FUNCTION_BLOCK FB_Component_SingleValve IMPLEMENTS I_Component
VAR_INPUT
	sName			: STRING[50];
	tTimeout		: TIME := T#0S;
END_VAR

VAR_IN_OUT
	bOutput			: BOOL;
END_VAR

VAR_OUTPUT
	bEnabled     	: BOOL;
	eState			: E_State := E_State.DISABLED;
	eNextState		: E_State := E_State.DISABLED;
	sStatusText 	: STRING[100];
END_VAR

VAR
	tTimeoutTimer	: TON;
	eLastState		: E_State;
END_VAR

VAR CONSTANT
	DISABLED		: E_State := E_State.DISABLED;
	READY			: E_State := E_State.READY;
	BUSY			: E_State := E_State.BUSY;
	HALTED			: E_State := E_State.HALTED;
	TIMEOUT			: E_State := E_State.TIMEOUT;
END_VAR

tTimeoutTimer(PT := tTimeout);

eState := eNextState;

CASE eState OF
	DISABLED: 	sStatusText := 'piston is disabled';
	READY: 		sStatusText := 'piston ready to operate';
	BUSY: 		sStatusText := 'piston busy';
	TIMEOUT:	sStatusText := 'piston in timeout';
				tTimeoutTimer(IN := TRUE);
				
				IF tTimeoutTimer.Q THEN
					tTimeoutTimer(IN := FALSE);
					eNextState := READY;
				END_IF
				
	HALTED:		sStatusText := 'piston halted';
END_CASE

METHOD M_Disable : BOOL
VAR_INPUT
END_VAR
IF eState = READY THEN
	bEnabled	:= FALSE;
	eNextState	:= DISABLED;
END_IF
END_METHOD

METHOD M_Enable : BOOL
VAR_INPUT
END_VAR
IF eState = DISABLED THEN
	bEnabled	:= TRUE;
	eNextState	:= READY;
END_IF
END_METHOD

METHOD M_Extend : BOOL
VAR_INPUT
END_VAR
IF eState = READY OR eState = BUSY THEN
	bOutput := TRUE;
END_IF
END_METHOD

METHOD M_Halt : BOOL
VAR_INPUT
END_VAR
IF eState <> HALTED AND eState <> DISABLED THEN
	eLastState := eState;
	eNextState := HALTED;
END_IF
END_METHOD

METHOD M_Resume : BOOL
VAR_INPUT
END_VAR
IF eState = HALTED THEN
	eNextState := eLastState;
END_IF
END_METHOD

METHOD M_Retract : BOOL
VAR_INPUT
END_VAR
IF eState = READY OR eState = BUSY THEN
	bOutput	:= FALSE;
END_IF
END_METHOD

END_FUNCTION_BLOCK

(* stored: Version 1.1.0.1, ProductVersion 3.1.4024.15
   POU FB_Component_SingleValve: Id {e241cca9-8ad1-4d32-953d-80e7ad832e70}, SpecialFunc None
   Method M_Disable: Id {1878d8e2-077c-448c-beb4-b9a7557014d9}
   Method M_Enable: Id {5cc8179e-f2ed-4378-940f-13b994787def}
   Method M_Extend: Id {452bb337-0657-46a1-ac4a-87cdd35da3f0}
   Method M_Halt: Id {6af66b53-6344-4d83-a0bf-1c140593c718}
   Method M_Resume: Id {3c239849-5b94-4c0a-a1a6-a48d6466116b}
   Method M_Retract: Id {8624003f-ef96-48fe-897d-ce8559b8e08c} *)
